FUNCTION_BLOCK Elevator
VAR_INPUT
END_VAR
VAR_OUTPUT
END_VAR
VAR
END_VAR

END_FUNCTION_BLOCK

(* stored: Version 1.1.0.1, ProductVersion 3.1.4024.2
   POU Elevator: Id {46ba5991-b5f9-4f5e-abab-a4ac0cc6420f}, SpecialFunc None *)
